# EPICS StreamDevice protocol: Sp2XXSup/sp2xx.proto
# SP2XX protocol file.

# Manuel specifies out terminator as "CR LF" but this creates errors when communicating with the device.

OutTerminator = CR;
InTerminator = "";

return = CR LF;
Stopped = $return ":";
Infusion = $return ">";
Withdrawal = $return "<";
NA = $return "NA";
na_or_blank = "%(\$1\$3){" $NA "|}"
ignored_status = $return "%*{:|>|<}";
rate_units = "{ml/m|ml/h|ul/m|ul/h}";
volume_units = "{ml|ul}";

mismatch_catcher {
	in $return "E";
	out "error?";
	in $return "%(\$1\$2)i" $ignored_status;
}

error_status {
	out "error?";
	in $return "%i" $ignored_status;
	@mismatch { mismatch_catcher; }
}

run {
    out "run";
	in "%(\$1\$3)#{" $NA "=0|" $Infusion "=1|" $Withdrawal "=1}";
	@mismatch { mismatch_catcher; }
}

run_status {
	out "run?";
	in "%{" $Stopped "|" $Infusion "|" $Withdrawal "}";
	@mismatch { mismatch_catcher; }
}

stop {
	out "stop";
	in "%(\$1\$3)#{" $NA "=0|" $Stopped "=1}";
	#@mismatch { mismatch_catcher; }
}

get_mode {
	out "mode?";
	in $return "%{IW|WI|I|W|CON}" $ignored_status;
	@mismatch { mismatch_catcher; }
}

set_mode {
	out "mode %{i\/w|w\/i|i|w|con}";
	in "%(\$1\$3)#{" $NA "=0|" $Stopped "=1}";
	@mismatch { mismatch_catcher; }
}

get_direction {
	out "dir?";
	in $return "%{I|W}" $ignored_status;
	@mismatch { mismatch_catcher; }
}

reverse_direction {
	out "dir rev";
	in $na_or_blank $ignored_status;
	@mismatch { mismatch_catcher; }
}

get_diam {
	out "dia?";
	in $return "%f" $ignored_status;
	@mismatch { mismatch_catcher; }
}

set_diam {
	out "dia %4.2f";
	in $na_or_blank $ignored_status;
	@mismatch { mismatch_catcher; }
}

get_voli {
	out "voli?";
	in $return "%f %(\$1\$3)" $volume_units $ignored_status;
	@mismatch { mismatch_catcher; }
}

set_voli {
	out "voli %05g %(\$1\$4)" $volume_units;
	in $na_or_blank $ignored_status;
	@mismatch { mismatch_catcher; }
}

get_volw {
	out "volw?";
	in $return "%f %(\$1\$3)" $volume_units $ignored_status;
	@mismatch { mismatch_catcher; }
}

set_volw {
	out "volw %05g %(\$1\$4)" $volume_units;
	in $na_or_blank $ignored_status;
	@mismatch { mismatch_catcher; }
}

get_ratew {
	out "ratew?";
	in $return "%f %(\$1\$3)" $rate_units $ignored_status;
	@mismatch { mismatch_catcher; }
}

set_ratew {
	out "ratew %05g %(\$1\$4)" $rate_units;
	in $na_or_blank $ignored_status;
	@mismatch { mismatch_catcher; }
}

get_ratei {
	out "ratei?";
	in $return "%f %(\$1\$3)" $rate_units $ignored_status;
	@mismatch { mismatch_catcher; }
}

set_ratei {
	out "ratei %05g %(\$1\$4)" $rate_units;
	in $na_or_blank $ignored_status;
	@mismatch { mismatch_catcher; }
}
